// TIA Portal V20 export
DATA_BLOCK "OperatorPrompts"   // DB123
// stored: Access Published, MemoryReserve 100
   VAR
      triggers { ExternalAccessible := 'False'; ExternalVisible := 'False'; ExternalWritable := 'False'} : Array[1..63] of Bool;
      activeOperatorPrompt { ExternalWritable := 'False'} : Int := 0;
      ack : Bool := FALSE;
   END_VAR
BEGIN
   triggers[1..63] := FALSE;
END_DATA_BLOCK
